TYPE ST_CX_EtherCATMasterPNetState :
STRUCT
	arrADSAddr		: ARRAY[0..5] OF BYTE;
	nPortNo			: UINT;
	arrAoeAddr		: ARRAY[0..5] OF BYTE;
	nDevState		: UINT;
	nPnIoError		: UINT;
	nPnIoDiag			: UINT;
END_STRUCT
END_TYPE

(* stored: Version 1.1.0.1, ProductVersion 3.1.4024.15
   DUT ST_CX_EtherCATMasterPNetState: Id {b8bafb88-5f08-4dc2-a7ec-618d2cbf8cc6} *)
